INTERFACE I_Collection EXTENDS I_Enumerable

METHOD AddItem : DINT
// Returns the index to which the new object is added into the list,
// or -1  to indicate that the object was not inserted
VAR_INPUT
    ipObject:       I_Object;
END_VAR
END_METHOD

METHOD Clear
// Remove all items from the list
VAR_INPUT
END_VAR
END_METHOD

METHOD Contains : BOOL
// Determines whether the list contains the querried object
VAR_INPUT
    ipObject:       I_Object;
END_VAR
END_METHOD

METHOD CopyToArray : BOOL
// Copies the whole list to a compatible one-dimensional array,
// starting at a specified index
VAR_IN_OUT
    aDest:          ARRAY [*] OF I_Object;
END_VAR
VAR_INPUT
    nIdx:           DINT;
END_VAR
END_METHOD

PROPERTY nCount : UDINT
GET
END_GET
END_PROPERTY

METHOD Remove : BOOL
// Remove the first occurerence of a specific object from the list
VAR_INPUT
    ipObject:       I_Object;
END_VAR
END_METHOD

END_INTERFACE

(* stored: Version 1.1.0.1, ProductVersion 3.1.4024.12
   Itf I_Collection: Id {57a1c343-f7a5-0e93-3b2c-627111f2aa09}
   Method AddItem: Id {278aeec7-af48-0b0a-2f2d-99b98cd1435c}
   Method Clear: Id {00c28f34-bd13-0119-0c75-c72092195800}
   Method Contains: Id {e324a86c-08eb-082c-0f99-c1ff9c7c3df6}
   Method CopyToArray: Id {1758ea08-9022-0973-3194-33e146e9bac3}
   Property nCount: Id {1d1d43a8-3c3c-067f-2ddc-54e64e241229}
   Get Get: Id {8f75c5e1-31e9-089c-08f2-b1d64ab1d1f5}
   Method Remove: Id {c9999731-75db-0087-1c58-bf38395be654} *)
